{attribute 'TcGenerated'}
// This function has been automatically generated from the project information.
VAR_GLOBAL CONSTANT
	{attribute 'const_non_replaced'}
	{attribute 'linkalways'}
	stLibVersion_TC3SafetyDiag : ST_LibVersion := (iMajor := 2, iMinor := 7, iBuild := 0, iRevision := 0, sVersion := '2.7.0');
END_VAR

(* stored: Version 1.1.0.1, ProductVersion 3.1.4022.12
   GVL Global_Version: Id {59efe83d-f4c1-4b2b-836c-45c104c390e5} *)
